{attribute wpf [Container(Layout.Wrap)]}
TYPE LayoutWrapStruct EXTENDS VariousTypesStruct :
STRUCT
END_STRUCT
END_TYPE

(* stored: Version 1.1.0.1, ProductVersion 3.1.4024.9
   DUT LayoutWrapStruct: Id {f3722166-5651-4e5a-b408-f54c82fb436d} *)
